# EPICS autosave request: iocBoot/generic_motors_ioc/dbSave/keithley_channel.req
%
% BURT Request File
%
% One Keithley
%
$(P)keithley$(D)
$(P)keithley$(D).DESC
$(P)keithley$(D):RqsGain
$(P)keithley$(D):RqsOffset
$(P)keithley$(D):RqsTime
